// TIA Portal V17 export
// export: Created 2025-03-07T09:16:32.6591916Z, ExportSetting WithDefaults, DisplayName Totally Integrated Automation Portal, DisplayVersion V17 Update 8, DisplayName TIA Portal Openness, DisplayVersion V17 Update 8, DisplayName TIA Portal Version Control Interface, DisplayVersion V17, DisplayName SINAMICS Startdrive Advanced, DisplayVersion V17 SP2, DisplayName SINAMICS Startdrive G110M, G120, G120C, G120D, G120P, G115D, DisplayVersion V17 SP2, DisplayName SINAMICS Startdrive G130, G150, S120, S150, SINAMICS MV, S210, DisplayVersion V17 SP2, DisplayName STEP 7 Professional, DisplayVersion V17 Update 8, DisplayName SINUMERIK ONE STEP 7 Toolbox, DisplayVersion V17 Update 12, DisplayName SINUMERIK 840D sl STEP 7 Toolbox, DisplayVersion V17 Update 12, DisplayName STEP 7 Safety, DisplayVersion V17 Update 6, DisplayName WinCC Advanced, DisplayVersion V17 Update 8
DATA_BLOCK "LBP_PowerrideConfig"   // DB78
TITLE = Configuration parameters of Powerride / Parámetros de configuración de powerride / Powerride Konfigurationsparameter
{ S7_Optimized_Access := 'FALSE'; DB_Accessible_From_OPC_UA := 'FALSE' }
AUTHOR : SINUMERIK
FAMILY : SINUMERIK_ONE
VERSION : 6.15
// Template with two predefined configurations for a Powerride / Plantilla con dos configuraciones predefinidas para un powerride / Vorlage mit zwei vordefinierten Konfigurationen für einen Powerride
// stored: AutoNumber false, DBAccessibleFromOPCUA false, DBAccessibleFromWebserver true, IsOnlyStoredInLoadMemory false, IsWriteProtectedInAS false
   VAR RETAIN
      configFeed { S7_SetPoint := 'True'} : "LBP_typePowerrideConfig";   // Konfiguration Vorschub % / configuration feed % / Configuración avance %
      configSpindle { S7_SetPoint := 'True'} : "LBP_typePowerrideConfig";   // Konfiguration Spindel % / configuration spindle % / Configuración husillo %
   END_VAR
BEGIN
   configFeed.pos100 := 19;
   configFeed.posMax := 23;
   configFeed.delay100 := T#500MS;
   configFeed.switchPos[2].value := 1;
   configFeed.switchPos[3].value := 2;
   configFeed.switchPos[4].value := 4;
   configFeed.switchPos[5].value := 6;
   configFeed.switchPos[6].value := 8;
   configFeed.switchPos[7].value := 10;
   configFeed.switchPos[8].value := 20;
   configFeed.switchPos[9].value := 30;
   configFeed.switchPos[10].value := 40;
   configFeed.switchPos[11].value := 50;
   configFeed.switchPos[12].value := 60;
   configFeed.switchPos[13].value := 70;
   configFeed.switchPos[14].value := 75;
   configFeed.switchPos[15].value := 80;
   configFeed.switchPos[16].value := 85;
   configFeed.switchPos[17].value := 90;
   configFeed.switchPos[18].value := 95;
   configFeed.switchPos[19].value := 100;
   configFeed.switchPos[20].value := 105;
   configFeed.switchPos[21].value := 110;
   configFeed.switchPos[22].value := 115;
   configFeed.switchPos[23..36].value := 120;
   configFeed.switchPos[2..18].ledColor := 7;
   configFeed.switchPos[19].ledColor := 2;
   configFeed.switchPos[20..22].ledColor := 3;
   configFeed.switchPos[23..36].ledColor := 1;
   configFeed.switchPos[1].vibrationIndex := 1;
   configFeed.switchPos[19].vibrationIndex := 2;
   configFeed.switchPos[23].vibrationIndex := 3;
   configSpindle.pos100 := 11;
   configSpindle.posMax := 15;
   configSpindle.delay100 := T#500MS;
   configSpindle.switchPos[1].value := 50;
   configSpindle.switchPos[2].value := 55;
   configSpindle.switchPos[3].value := 60;
   configSpindle.switchPos[4].value := 65;
   configSpindle.switchPos[5].value := 70;
   configSpindle.switchPos[6].value := 75;
   configSpindle.switchPos[7].value := 80;
   configSpindle.switchPos[8].value := 85;
   configSpindle.switchPos[9].value := 90;
   configSpindle.switchPos[10].value := 95;
   configSpindle.switchPos[11].value := 100;
   configSpindle.switchPos[12].value := 105;
   configSpindle.switchPos[13].value := 110;
   configSpindle.switchPos[14].value := 115;
   configSpindle.switchPos[15..36].value := 120;
   configSpindle.switchPos[1..10].ledColor := 7;
   configSpindle.switchPos[11].ledColor := 2;
   configSpindle.switchPos[12..14].ledColor := 3;
   configSpindle.switchPos[15..36].ledColor := 1;
   configSpindle.switchPos[11].vibrationIndex := 2;
   configSpindle.switchPos[15].vibrationIndex := 3;
   configSpindle.switchPos[23].vibrationIndex := 3;
END_DATA_BLOCK
